{attribute 'qualified_only'}
VAR_GLOBAL
	ScadaInterface: MainInterface;
END_VAR

(* stored: Version 1.1.0.1, ProductVersion 3.1.4024.4
   GVL Interfacex: Id {a0873a74-9354-45d6-8d35-c920e367cf21} *)
